TYPE ST_HMI_Machine_Config :
STRUCT
END_STRUCT
END_TYPE

(* stored: Version 1.1.0.1, ProductVersion 3.1.4024.12
   DUT ST_HMI_Machine_Config: Id {7dbbc7b7-8c48-46e2-ad35-edc3e2719b2b} *)
